FUNCTION_BLOCK FB_ADSCommunicationStatus
VAR_INPUT
	Timeout	:	TIME := T#1S;
	LocalAdsPort	:	T_AmsPort;
END_VAR
VAR
	instReadLocalAMSNetId	:	FB_GetLocalAmsNetId;
	statExecuteReadingLocalAMSNetId	:	BOOL := TRUE;
	statBusyReadLocalAMSNetId	:	BOOL;
	statErrorReadLocalAMSNetId	:	BOOL;
	statErrorNumberReadLocalAMSNetId	:	UDINT;
	statReadLocalAMSNetId	:	T_AmsNetID;
	statReadLocalAMSNetIdSeprated	:	T_AmsNetIdArr;
	
	statGettingIpAddress	:	BOOL;
	statLocalIpAddress	:	STRING;
	
	instReadADSState	:	ADSRDSTATE;
	statExecuteReadingAdsState	:	BOOL;
	statBusyReadAdsState	:	BOOL;
	statErrorReadAdsState	:	BOOL;
	statErrorNumberAdsState	:	UDINT;
	statReadAdsState	:	UDINT;
END_VAR

(*===================== Reading local AMSNetId =====================*)
instReadLocalAMSNetId(bExecute := statExecuteReadingLocalAMSNetId,
					  tTimeOut := Timeout,
					  bBusy => statBusyReadLocalAMSNetId,
					  bError => statErrorReadLocalAMSNetId,
					  nErrId => statErrorNumberReadLocalAMSNetId,
					  AddrString => statReadLocalAMSNetId,
					  AddrBytes => statReadLocalAMSNetIdSeprated);
					  
IF NOT statBusyReadLocalAMSNetId AND NOT statErrorReadLocalAMSNetId AND
	statExecuteReadingLocalAMSNetId THEN
	statExecuteReadingLocalAMSNetId := FALSE;
	statGettingIpAddress := TRUE;
	statExecuteReadingAdsState := TRUE;
END_IF

(*===================== Reading local AMSNetId =====================*)
IF statGettingIpAddress THEN
	statLocalIpAddress := GetDeviceIpAddress(statReadLocalAMSNetIdSeprated);
	statGettingIpAddress := FALSE;
END_IF

(*===================== Reading Ads state =====================*)
instReadADSState(NETID := statReadLocalAMSNetId,
				 PORT := LocalAdsPort,
				 RDSTATE := statExecuteReadingAdsState,
			     TMOUT := Timeout,
				 BUSY => statBusyReadAdsState,
				 ERR => statErrorReadAdsState,
				 ERRID => statErrorNumberAdsState,
				 ADSSTATE => statReadAdsState);
					  
IF NOT statBusyReadAdsState AND NOT statErrorReadAdsState AND
	statExecuteReadingAdsState THEN
	statExecuteReadingAdsState := FALSE;
END_IF

METHOD PRIVATE GetDeviceIpAddress : String
VAR_INPUT
	CurrentAMSNetId	:	T_AmsNetIdArr;
END_VAR
VAR
	tempRunCounter	:	INT;
	tempIpAddressConverted	:	STRING;
END_VAR
FOR tempRunCounter := 0 TO 3 DO
	tempIpAddressConverted := CONCAT(tempIpAddressConverted, BYTE_TO_STRING(CurrentAMSNetId[tempRunCounter]));
	IF tempRunCounter < 3 THEN
		tempIpAddressConverted := CONCAT(tempIpAddressConverted, '.');
	END_IF
END_FOR

GetDeviceIpAddress := tempIpAddressConverted;
END_METHOD

PROPERTY PUBLIC LocalAMSNetId : String
GET
LocalAMSNetId := statReadLocalAMSNetId;
END_GET
END_PROPERTY

PROPERTY PUBLIC LocalIpAddress : String
GET
LocalIpAddress := statLocalIpAddress;
END_GET
END_PROPERTY

END_FUNCTION_BLOCK

(* stored: Version 1.1.0.1
   POU FB_ADSCommunicationStatus: Id {fc26bda7-2b0c-49ee-914f-e68b93c48878}, SpecialFunc None
   Method GetDeviceIpAddress: Id {6b460412-9514-4e9a-b6c9-8eebbe2fbb84}
   Property LocalAMSNetId: Id {7b71f754-a9bd-4d11-a914-4354786a1931}
   Get Get: Id {219b9a17-cb1d-486e-8706-680f14c1b592}
   Property LocalIpAddress: Id {6000413c-bfbf-43ca-8c0b-09816ce2d821}
   Get Get: Id {020ecc30-ae91-4c39-9568-5747342c3c80} *)
